TYPE "MEStoPLC_MainCheckIn_ext"
VERSION : 0.1
   STRUCT
      Load_Station1PartOK : Bool;
      Load_Station1PartNG : Bool;
      Load_Station1ReqMesDone : Bool;
      Load_Station1Spare : Bool;
      Load_Station1Spare1 : Bool;
      Load_Station1Spare2 : Bool;
      Load_Station1Spare3 : Bool;
      Load_Station1Spare4 : Bool;
      Load_Station2PartOK : Bool;
      Load_Station2PartNG : Bool;
      Load_Station2ReqMesDone : Bool;
      Load_Station2Spare : Bool;
      Load_Station2Spare1 : Bool;
      Load_Station2Spare2 : Bool;
      Load_Station2Spare3 : Bool;
      Load_Station2Spare4 : Bool;
      Load_Station3PartOK : Bool;
      Load_Station3PartNG : Bool;
      Load_Station3ReqMesDone : Bool;
      Load_Station3Spare : Bool;
      Load_Station3Spare1 : Bool;
      Load_Station3Spare2 : Bool;
      Load_Station3Spare3 : Bool;
      Load_Station3Spare4 : Bool;
      Load_Station4PartOK : Bool;
      Load_Station4PartNG : Bool;
      Load_Station4ReqMesDone : Bool;
      Load_Station4Spare : Bool;
      Load_Station4Spare1 : Bool;
      Load_Station4Spare2 : Bool;
      Load_Station4Spare3 : Bool;
      Load_Station4Spare4 : Bool;
      Load_Station5PartOK : Bool;
      Load_Station5PartNG : Bool;
      Load_Station5ReqMesDone : Bool;
      Load_Station5Spare : Bool;
      Load_Station5Spare1 : Bool;
      Load_Station5Spare2 : Bool;
      Load_Station5Spare3 : Bool;
      Load_Station5Spare4 : Bool;
      Load_Station6PartOK : Bool;
      Load_Station6PartNG : Bool;
      Load_Station6ReqMesDone : Bool;
      Load_Station6Spare : Bool;
      Load_Station6Spare1 : Bool;
      Load_Station6Spare2 : Bool;
      Load_Station6Spare3 : Bool;
      Load_Station6Spare4 : Bool;
      Load_Station7PartOK : Bool;
      Load_Station7PartNG : Bool;
      Load_Station7ReqMesDone : Bool;
      Load_Station7Spare : Bool;
      Load_Station7Spare1 : Bool;
      Load_Station7Spare2 : Bool;
      Load_Station7Spare3 : Bool;
      Load_Station7Spare4 : Bool;
      Load_Station8PartOK : Bool;
      Load_Station8PartNG : Bool;
      Load_Station8ReqMesDone : Bool;
      Load_Station8Spare : Bool;
      Load_Station8Spare5 : Bool;
      Load_Station8Spare6 : Bool;
      Load_Station8Spare8 : Bool;
      Load_Station8Spare9 : Bool;
   END_STRUCT;

END_TYPE

